PROGRAM MAIN
VAR
	FB_TEST : FB_FruitTemperatureControl;
END_VAR

FB_TEST(//Input
		eControlMode := GVL.eTestMode,
		fTfruitRef := GVL.fTestTfruitRef,
		fTthermostat := GVL.fTestTthermostat,
		fTfruit := GVL.fTestTfruit,
		fKp := GVL.fTestKp,
		fKi := GVL.tTestKi,
		fKt := GVL.tTestKt,
		bReset := GVL.bTestReset,
		
		//Output
		fTthermostatOut => GVL.fTestTthermostatOut,
		sStateText => GVL.sTestStateText,
		bRelay => GVL.bRelay,
		
		//Test output
		fTestUantiWind => GVL.fTestUantiWind,
		fTestUerrorSat => GVL.fTestUerrorSat,
		fTestUvoorSat => GVL.fTestUvoorSat,
		fTestTsetOut => GVL.fTestTsetOut);

END_PROGRAM

(* stored: Version 1.1.0.1, ProductVersion 3.1.4024.11
   POU MAIN: Id {a1204864-8e37-4b95-b4e1-eee49f101afa}, SpecialFunc None *)
